(* CoDeSys 2.3 export: all2.exp *)
(* Libraries: ANALYZATION.LIB 5.10.99 09:05:06, ComService.lib 21.5.09 14:28:28, IECSFC.LIB 13.4.06 15:51:28, modbus.lib 27.5.09 09:22:38, STANDARD.LIB 4.10.05 11:14:46, SysLibCom.lib 20.2.06 12:31:08 *)

(* PLC configuration (modules and I/O channels)
PLC110_30 [Root] node -1, in %IB0 out %QB0 {param 1 = PLC110-30_v2; param 2 = 1; param 3 = 1000}
  Fast discrete inputs [I_SIMPLE_INPUT] node 0, in %IB0 out %QB0 {param 1 = Fast discrete inputs; param 2 = 10000}
    AT %IX0.0 [BitInput] Дискретный вход 1 {param 1 = Enter name}
    AT %IX0.1 [BitInput] Дискретный вход 2 {param 1 = Enter name}
  Дискретные входы - 16 [ID130] node 1, in %IB1 out %QB1 {param 1 = Дискретные входы; param 2 = 10; param 3 = 16}
    AT %IB1.0 [ByteInput] 8 дискретных входов {param 1 = Enter name}
    AT %IB1.1 [ByteInput] 8 дискретных входов {param 1 = Enter name}
  Быстрые дискретные выходы [OWEN_ID570] node 2, in %IB2 out %QB2 {param 1 = Быстрые дискретные выходы; param 2 = FALSE; param 3 = FALSE; param 4 = FALSE; param 5 = FALSE}
    AT %QX2.0 [BitOutput] Быстрый дискретный выход 1 {param 1 = Enter name}
    AT %QX2.1 [BitOutput] Быстрый дискретный выход 2 {param 1 = Enter name}
    AT %QX2.2 [BitOutput] Быстрый дискретный выход 3 {param 1 = Enter name}
    AT %QX2.3 [BitOutput] Быстрый дискретный выход 4 {param 1 = Enter name}
  Дискретные выходы - 8 [ID131] node 3, in %IB3 out %QB3 {param 1 = Дискретные выходы; param 2 = 0; param 3 = No; param 4 = 10}
    AT %QB3.0 [ByteOutput] 8 дискретных выходов {param 1 = Enter name}
  Специальный вход [ID103] node 4, in %IB4 out %QB4 {param 1 = Специальный вход}
    AT %IX4.0 [BitInput] Специальный вход {param 1 = Enter name}
  Специальный выход [ID104] node 5, in %IB5 out %QB5 {param 1 = Специальный выход}
    AT %QX5.0 [BitOutput] Специальный выход {param 1 = Enter name}
  ModBus (Master) [MODBUS_MASTER_ID450] node 6, in %IB6 out %QB6 {param 1 = ModBus (Master); param 2 = No}
    AT %QD6.0 [DWordOutput] Last address {param 1 = Enter name}
    AT %QW6.1 [WordOutput] Last error {param 1 = Enter name}
    RS-485-1 [COM1_USART] node 0, in %IB6.0 out %QB6.0 {param 1 = RS-485-1; param 2 = 9600; param 3 = NO PARITY CHECK; param 4 = 8 bits; param 5 = One stop bit; param 6 = RS485; param 7 = ASCII; param 8 = 0; param 9 = No}
*)

(* Global variable list: Global_Variables *)
VAR_GLOBAL
    (* Fast discrete inputs (encoder) *)
    gEncoderA   AT %IX0.0 : BOOL;    (* DI1 - Encoder A (fast input) *)
    gEncoderB   AT %IX0.1 : BOOL;    (* DI2 - Encoder B (fast input) *)

    (* ModBus (Master) system/channel variables exposed by device configuration *)
    gModbus_Master_Channel AT %QD6.0 : DWORD; (* ModBus Master: channel/last address (Q area) *)
    gModbus_Master_LastError AT %QW6.1 : WORD; (* ModBus Master: last error code (Q area) *)

    (* Discrete inputs (DI3..DI18) mapped to %IX1.0.0 - %IX1.1.7 *)
    gDI_3  AT %IX1.0.0 : BOOL; (* DI3 *)
    gDI_4  AT %IX1.0.1 : BOOL; (* DI4 *)
    gDI_5  AT %IX1.0.2 : BOOL; (* DI5 *)
    gDI_6  AT %IX1.0.3 : BOOL; (* DI6 *)
    gDI_7  AT %IX1.0.4 : BOOL; (* DI7 *)
    gDI_8  AT %IX1.0.5 : BOOL; (* DI8 *)
    gDI_9  AT %IX1.0.6 : BOOL; (* DI9 *)
    gDI_10 AT %IX1.0.7 : BOOL; (* DI10 *)
    gDI_11 AT %IX1.1.0 : BOOL; (* DI11 *)
    gDI_12 AT %IX1.1.1 : BOOL; (* DI12 *)
    gDI_13 AT %IX1.1.2 : BOOL; (* DI13 *)
    gDI_14 AT %IX1.1.3 : BOOL; (* DI14 *)
    gDI_15 AT %IX1.1.4 : BOOL; (* DI15 *)
    gDI_16 AT %IX1.1.5 : BOOL; (* DI16 *)
    gDI_17 AT %IX1.1.6 : BOOL; (* DI17 *)
    gDI_18 AT %IX1.1.7 : BOOL; (* DI18 *)

    (* Discrete outputs - relay DO1..DO8 mapped to %QX3.0.0..%QX3.0.7 *)
    gDO_1 AT %QX3.0.0 : BOOL;  (* DO1 - Forward *)
    gDO_2 AT %QX3.0.1 : BOOL;  (* DO2 - Reverse *)
    gDO_3 AT %QX3.0.2 : BOOL;  (* DO3 - In position indicator *)
    gDO_4 AT %QX3.0.3 : BOOL;  (* DO4 *)
    gDO_5 AT %QX3.0.4 : BOOL;  (* DO5 *)
    gDO_6 AT %QX3.0.5 : BOOL;  (* DO6 *)
    gDO_7 AT %QX3.0.6 : BOOL;  (* DO7 *)
    gDO_8 AT %QX3.0.7 : BOOL;  (* DO8 *)

    (* Fast/transistor discrete outputs DO9..DO12 mapped to %QX2.0..%QX2.3 (fast outputs module) *)
    gDO_9  AT %QX2.0 : BOOL; (* DO9  - fast/transistor output *)
    gDO_10 AT %QX2.1 : BOOL; (* DO10 *)
    gDO_11 AT %QX2.2 : BOOL; (* DO11 *)
    gDO_12 AT %QX2.3 : BOOL; (* DO12 *)

    (* Variables for Modbus and internal state (no AT) *)
    (*
        Modbus (holding) register map served by ESP (slave):
        Register numbers (offset 0):
        0-1   : target angle (REAL)            (REG_TARGET_ANGLE_HI/LO)
        2-3   : current angle (REAL)           (REG_CURRENT_ANGLE_HI/LO)
        4-5   : reserved
        6     : status (WORD)                  (0=Stop,1=Moving,2=In position)
        7     : error code (WORD)
        8     : command (WORD)                 (1=Start,2=Stop,3=Calib)
        9-10  : encoder count (DINT, hi/lo)
        11    : PPR (WORD)
        12    : quad mode (WORD)
        13    : max time (WORD)
        14-15 : hysteresis (REAL)
    *)
    gTargetAngle : REAL := 45.0;    (* target angle, degrees *)
    gCurrentAngle : REAL := 0.0;    (* current angle, degrees *)
    gAngleFromStart : REAL := 0.0;  (* angle from program start *)
    gStatus : INT := 0;             (* 0=Stop,1=Moving,2=In position *)
    gErrorCode : INT := 0;          (* 0=OK,1=Timeout,2=Fault *)
    gCommand : INT := 0;            (* 1=Start,2=Stop,3=Calibrate *)
    gEncoderCount : DINT := 0;     (* encoder counter for Modbus *)

    (* Calibration / Modbus helper variables *)
    gStartCalib : BOOL := FALSE;
    gCalibRunning : BOOL := FALSE;
    gCalibStatus : INT := 0;
    gCalibRevsDone : INT := 0;
    gCalibRevsTarget : INT := 3;
    gCalibMeasured : REAL := 0.0;
    gCalibCountsPerRev : DINT := 0;
END_VAR

(* Data type *)
(* Local fallback: COMSETTINGS_FALLBACK - avoids collision with SysLibCom.lib when library types are not exposed to the IDE. Remove this TYPE when real `COMSETTINGS` is available. *)
TYPE COMSETTINGS_FALLBACK : STRUCT
    Port : INT;
    dwBaudRate : DWORD;
    byStopBits : BYTE;
    byParity : BYTE;
    dwTimeout : DWORD;
    dwBufferSize : DWORD;
    dwScan : DWORD;
END_STRUCT
END_TYPE
PROGRAM PLC_PRG
VAR
    (* Encoder / positioning parameters and state *)
    COUNTS_PER_REV : INT := 360;
    ANGLE_PER_COUNT : REAL := 1.0;
    HYSTERESIS : REAL := 1.5;
    MAX_MOVE_TIME : INT := 3000;

    encoderCount : DINT := 0;
    prevEncoderA : BOOL := FALSE;

    gLocalTargetAngle : REAL := 0.0; (* local copy of target from Modbus *)

    motorFwd : BOOL := FALSE;
    motorRev : BOOL := FALSE;
    isPositioned : BOOL := FALSE;
    moveTimer : INT := 0;

    (* Modbus / COM-service variables (library types) *)
    Settings : COMSETTINGS_FALLBACK; (* fallback type when SysLibCom.lib types are not visible; replace with COMSETTINGS if library exports it *)
    COM_SERVICE1 : COM_SERVICE; (* ComService.lib FB instance *)
    getHold : MB_RD_HOLD_REGS; (* modbus.lib FB instance for Read Holding Registers *)

    Buffer : ARRAY[0..255] OF BYTE;
    cmpl : BOOL;
    excep : BYTE;
    DataSize : WORD;
    TimeOut : TIME := T#50ms;
    port_opened : BYTE := 0; (* 0=closed,2=opened *)
    enabl : BOOL := TRUE; (* enable for modbus FBs *)

    (* local temporaries used to unpack returned registers *)
    tmp_dw : DWORD;
    tmpFloat : REAL;
    tmpHi : WORD;
    tmpLo : WORD;
    tmpDiff : REAL := 0.0; (* local diff variable declared here *)
END_VAR
